PROGRAM Reaktoranlage
VAR
	R1				:FB_Reaktoreinheit;
	R2				:FB_Reaktoreinheit;
	
	// Instanziierung von Switchfunktion für Update-Variable
	Switch_R1		:FB_UpdateHandler;
	Switch_R2		:FB_UpdateHandler;
	Switch_R3		:FB_UpdateHandler;
	Switch_R4		:FB_UpdateHandler;
	Switch_R5		:FB_UpdateHandler;
	Switch_R6		:FB_UpdateHandler;
	Switch_R7		:FB_UpdateHandler;
END_VAR

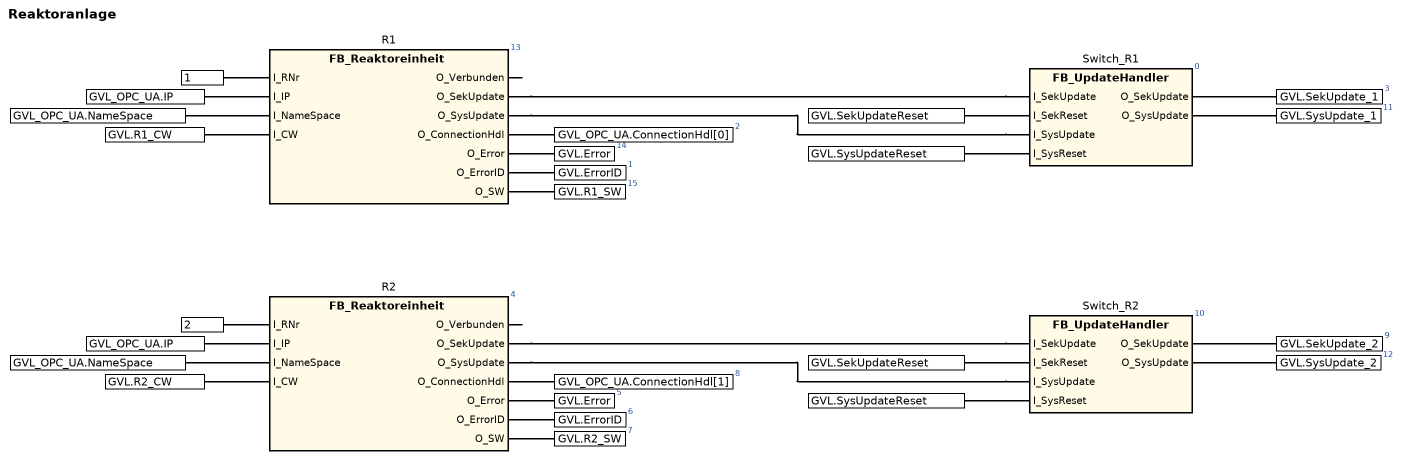
Switch_R1(
    I_SekUpdate := R1.O_SekUpdate,
    I_SekReset := GVL.SekUpdateReset,
    I_SysUpdate := R1.O_SysUpdate,
    I_SysReset := GVL.SysUpdateReset); // FB_UpdateHandler
GVL.ErrorID := R1.O_ErrorID;
GVL_OPC_UA.ConnectionHdl[0] := R1.O_ConnectionHdl;
GVL.SekUpdate_1 := Switch_R1.O_SekUpdate;
R2(I_RNr := 2, I_IP := GVL_OPC_UA.IP, I_NameSpace := GVL_OPC_UA.NameSpace, I_CW := GVL.R2_CW); // FB_Reaktoreinheit
GVL.Error := R2.O_Error;
GVL.ErrorID := R2.O_ErrorID;
GVL.R2_SW := R2.O_SW;
GVL_OPC_UA.ConnectionHdl[1] := R2.O_ConnectionHdl;
GVL.SekUpdate_2 := Switch_R2.O_SekUpdate;
Switch_R2(
    I_SekUpdate := R2.O_SekUpdate,
    I_SekReset := GVL.SekUpdateReset,
    I_SysUpdate := R2.O_SysUpdate,
    I_SysReset := GVL.SysUpdateReset); // FB_UpdateHandler
GVL.SysUpdate_1 := Switch_R1.O_SysUpdate;
GVL.SysUpdate_2 := Switch_R2.O_SysUpdate;
R1(I_RNr := 1, I_IP := GVL_OPC_UA.IP, I_NameSpace := GVL_OPC_UA.NameSpace, I_CW := GVL.R1_CW); // FB_Reaktoreinheit
GVL.Error := R1.O_Error;
GVL.R1_SW := R1.O_SW;

END_PROGRAM

(* stored: Version 1.1.0.1, ProductVersion 3.1.4024.12
   POU Reaktoranlage: Id {940c7541-d79f-49db-a967-8e3935b5d8ed}, SpecialFunc None *)
